// TIA Portal project "S71200OPCUA" (V16)

(* hardware
DEVICE "S7-1200 station_1"  S7-1200 Station
   slot 0: "Rack_0"  S7-1200 Rack  Rack  V1.0
   slot 1: "PLC_1"  CPU 1212C AC/DC/Rly  6ES7 212-1BE40-0XB0  V4.4
*)

// ===== PLC "PLC_1"  CPU 1212C AC/DC/Rly =====

VAR_GLOBAL   // PLC tag table "Default tag table"
   "Clock_Byte" AT %MB0 : Byte;
   "Clock_10Hz" AT %M0.0 : Bool;
   "Clock_5Hz" AT %M0.1 : Bool;
   "Clock_2.5Hz" AT %M0.2 : Bool;
   "Clock_2Hz" AT %M0.3 : Bool;
   "Clock_1.25Hz" AT %M0.4 : Bool;
   "Clock_1Hz" AT %M0.5 : Bool;
   "Clock_0.625Hz" AT %M0.6 : Bool;
   "Clock_0.5Hz" AT %M0.7 : Bool;
   "Disconnect" AT %M10.0 : Bool;
   "I_Sensor" AT %I10.0 : Bool;
   "Q_Speed" AT %QD100 : Real;
   "I_Boxdetected" AT %I10.1 : Bool;
   "I_PosX" AT %ID100 : Real;
   "I_PosY" AT %ID104 : Real;
   "I_PosZ" AT %ID108 : Real;
   "Q_PosX" AT %QD104 : Real;
   "Q_PosY" AT %QD108 : Real;
   "Q_PosZ" AT %QD112 : Real;
   "Q_Vacuum" AT %Q10.0 : Bool;
   "I_Flow" AT %ID112 : Real;
   "I_Level" AT %ID116 : Real;
   "Q_Filling" AT %QD116 : Real;
   "Q_Draining" AT %QD120 : Real;
   "I_Diffuse2m(1)" AT %I10.2 : Bool;
   "I_Diffuse2m(2)" AT %I10.3 : Bool;
   "Q_Conveyor2m(1)" AT %Q10.1 : Bool;
   "Q_Conveyor2m(2)" AT %Q10.2 : Bool;
END_VAR

DATA_BLOCK "OPC"   // DB1
{ S7_Optimized_Access := 'TRUE' }
VERSION : 0.1
   VAR
      Tank : Struct
         I_Level : Real;
         I_Flow : Real;
         Q_Filling : Real;
         Q_Draining : Real;
      END_STRUCT;
      Conveyor : Struct
         Q_Conveyor : Bool;
         "I_Sensor2m(1)" : Bool;
         "I_Sensor2m(2)" : Bool;
         "Q_Conveyor2m(1)" : Bool;
         "Q_Conveyor2m(2)" : Bool;
         I_Start : Bool;
         I_Stop : Bool;
         Q_Speed : Real;
         I_Sensor : Bool;
         Q_BoxCount : DInt;
         I_Reset : Bool;
         I_Maxlimit : Real := 6.0;
         I_Minlimit : Real := 2.0;
         I_Speed : Real := 1.0;
      END_STRUCT;
      "Pick and Place axis" : Struct
         I_Tolerance : Real := 0.02;
         IQ_Step : Int;
         I_Start : Bool;
         I_Init : Bool;
         I_XPos : Real;
         I_YPos : Real;
         I_ZPos : Real;
         I_BoxDetect : Bool;
         Q_XPos : Real;
         Q_YPos : Real;
         Q_ZPos : Real;
         Q_Vacuum : Bool;
         Q_Placed : Bool;
         Pos1 : Struct
            X : Real := 2.7;
            Y : Real := 3.9;
            Z : Real := 5.0;
         END_STRUCT;
         Pos2 : Struct
            X : Real := 6.6;
            Y : Real := 3.3;
            Z : Real := 4.2;
         END_STRUCT;
      END_STRUCT;
      Process : Struct
         I_Start : Bool;
         I_Stop : Bool;
         Process : Bool;
      END_STRUCT;
   END_VAR
BEGIN
END_DATA_BLOCK

// folder: 3Axis

DATA_BLOCK "Axis_DB"   // DB4
{ S7_Optimized_Access := 'TRUE' }
VERSION : 0.1
// stored: InstanceOfName Axis
"Axis"
BEGIN
END_DATA_BLOCK

// folder: Conveyor

DATA_BLOCK "IEC_Counter_0_DB"   // DB2
{ S7_Optimized_Access := 'TRUE' }
AUTHOR : Simatic
FAMILY : IEC
NAME : CNTR
VERSION : 1.0
// stored: InstanceOfName IEC_COUNTER
"IEC_COUNTER"
BEGIN
END_DATA_BLOCK

DATA_BLOCK "Conveyor_DB_1"   // DB5
{ S7_Optimized_Access := 'TRUE' }
VERSION : 0.1
// stored: InstanceOfName Conveyor
"Conveyor"
BEGIN
END_DATA_BLOCK

// folder: System blocks/Program resources

DATA_BLOCK "IEC_Timer_0_DB_1"   // DB3
{ S7_Optimized_Access := 'TRUE' }
AUTHOR : Simatic
FAMILY : IEC
NAME : IEC_TMR
VERSION : 1.0
// stored: InstanceOfName IEC_TIMER
"IEC_TIMER"
BEGIN
END_DATA_BLOCK

DATA_BLOCK "IEC_Timer_0_DB"   // DB6
{ S7_Optimized_Access := 'TRUE' }
AUTHOR : Simatic
FAMILY : IEC
NAME : IEC_TMR
VERSION : 1.0
// stored: InstanceOfName IEC_TIMER
"IEC_TIMER"
BEGIN
END_DATA_BLOCK

DATA_BLOCK "IEC_Timer_0_DB_2"   // DB7
{ S7_Optimized_Access := 'TRUE' }
AUTHOR : Simatic
FAMILY : IEC
NAME : IEC_TMR
VERSION : 1.0
// stored: InstanceOfName IEC_TIMER
"IEC_TIMER"
BEGIN
END_DATA_BLOCK

// folder: (top level)

ORGANIZATION_BLOCK "Main"   // OB1, FBD, ProgramCycle
TITLE = "Main Program Sweep (Cycle)"
{ S7_Optimized_Access := 'TRUE' }
VERSION : 0.1
   VAR_INPUT
      Initial_Call : Bool;   // Initial call of this OB
      Remanence : Bool;   // =True, if remanent data are available
   END_VAR
BEGIN

REGION Network 1: Process
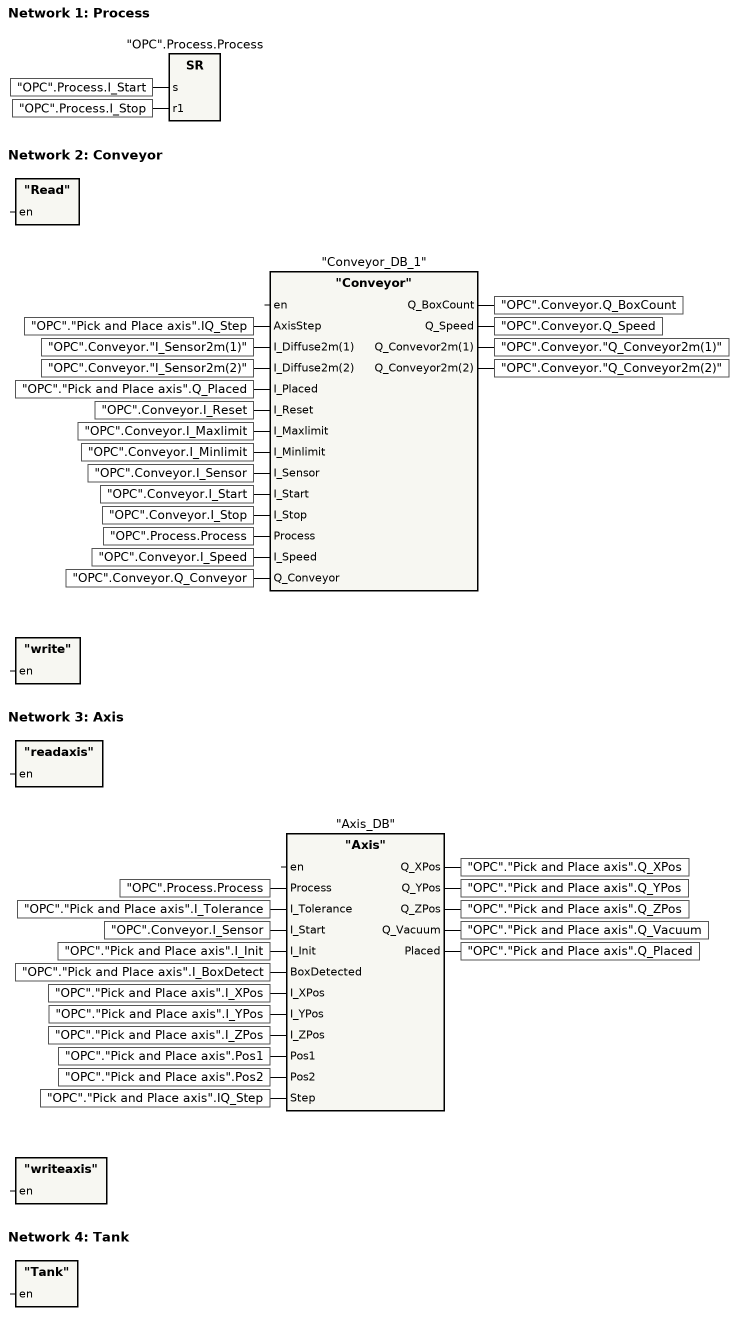
   IF "OPC".Process.I_Start THEN
       "OPC".Process.Process := TRUE;   // SR flip-flop
   END_IF;
   IF "OPC".Process.I_Stop THEN "OPC".Process.Process := FALSE; END_IF;
END_REGION

REGION Network 2: Conveyor
   "Read"();
   "Conveyor_DB_1"(AxisStep := "OPC"."Pick and Place axis".IQ_Step,   // "Conveyor"
                   "I_Diffuse2m(1)" := "OPC".Conveyor."I_Sensor2m(1)",
                   "I_Diffuse2m(2)" := "OPC".Conveyor."I_Sensor2m(2)",
                   I_Placed := "OPC"."Pick and Place axis".Q_Placed,
                   I_Reset := "OPC".Conveyor.I_Reset,
                   I_Maxlimit := "OPC".Conveyor.I_Maxlimit,
                   I_Minlimit := "OPC".Conveyor.I_Minlimit,
                   I_Sensor := "OPC".Conveyor.I_Sensor,
                   I_Start := "OPC".Conveyor.I_Start,
                   I_Stop := "OPC".Conveyor.I_Stop,
                   Process := "OPC".Process.Process,
                   I_Speed := "OPC".Conveyor.I_Speed,
                   Q_Conveyor := "OPC".Conveyor.Q_Conveyor,
                   Q_BoxCount => "OPC".Conveyor.Q_BoxCount,
                   Q_Speed => "OPC".Conveyor.Q_Speed,
                   "Q_Convevor2m(1)" => "OPC".Conveyor."Q_Conveyor2m(1)",
                   "Q_Conveyor2m(2)" => "OPC".Conveyor."Q_Conveyor2m(2)");
   "write"();
END_REGION

REGION Network 3: Axis
   "readaxis"();
   "Axis_DB"(Process := "OPC".Process.Process,   // "Axis"
             I_Tolerance := "OPC"."Pick and Place axis".I_Tolerance,
             I_Start := "OPC".Conveyor.I_Sensor,
             I_Init := "OPC"."Pick and Place axis".I_Init,
             BoxDetected := "OPC"."Pick and Place axis".I_BoxDetect,
             I_XPos := "OPC"."Pick and Place axis".I_XPos,
             I_YPos := "OPC"."Pick and Place axis".I_YPos,
             I_ZPos := "OPC"."Pick and Place axis".I_ZPos,
             Pos1 := "OPC"."Pick and Place axis".Pos1,
             Pos2 := "OPC"."Pick and Place axis".Pos2,
             "Step" := "OPC"."Pick and Place axis".IQ_Step,
             Q_XPos => "OPC"."Pick and Place axis".Q_XPos,
             Q_YPos => "OPC"."Pick and Place axis".Q_YPos,
             Q_ZPos => "OPC"."Pick and Place axis".Q_ZPos,
             Q_Vacuum => "OPC"."Pick and Place axis".Q_Vacuum,
             Placed => "OPC"."Pick and Place axis".Q_Placed);
   "writeaxis"();
END_REGION

REGION Network 4: Tank
   "Tank"();
END_REGION
END_ORGANIZATION_BLOCK

// folder: 3Axis

FUNCTION_BLOCK "Axis"   // FB3, FBD
{ S7_Optimized_Access := 'TRUE' }
VERSION : 0.1
   VAR_INPUT
      Process : Bool;
      I_Tolerance : Real;
      I_Start : Bool;
      I_Init : Bool;
      BoxDetected : Bool;
      I_XPos : Real;
      I_YPos : Real;
      I_ZPos : Real;
      Pos1 : Struct
         X : Real;
         Y : Real;
         Z : Real;
      END_STRUCT;
      Pos2 : Struct
         X : Real;
         Y : Real;
         Z : Real;
      END_STRUCT;
   END_VAR
   VAR_OUTPUT
      Q_XPos : Real;
      Q_YPos : Real;
      Q_ZPos : Real;
      Q_Vacuum : Bool;
      Placed : Bool;
   END_VAR
   VAR_IN_OUT
      "Step" : Int;
   END_VAR
   VAR
      PosX1Min : Real;
      PosX1Max : Real;
      PosY1Min : Real;
      PosY1Max : Real;
      PosZ1Min : Real;
      PosZ1Max : Real;
      PosX2Min : Real;
      PosX2Max : Real;
      PosY2Min : Real;
      PosY2Max : Real;
      PosZ2Min : Real;
      PosZ2Max : Real;
   END_VAR
   VAR_TEMP   // added for the SCL form of the ladder/FBD networks
      _w1 : Bool;
   END_VAR
BEGIN

REGION Network 1: Position Tolerance P1
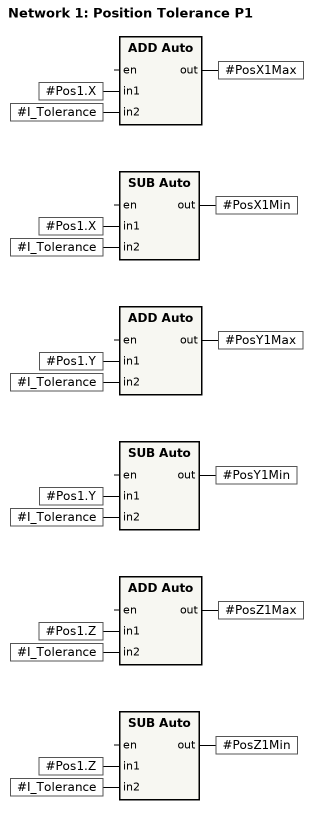
   #PosX1Max := #Pos1.X + #I_Tolerance;
   #PosX1Min := #Pos1.X - #I_Tolerance;
   #PosY1Max := #Pos1.Y + #I_Tolerance;
   #PosY1Min := #Pos1.Y - #I_Tolerance;
   #PosZ1Max := #Pos1.Z + #I_Tolerance;
   #PosZ1Min := #Pos1.Z - #I_Tolerance;
END_REGION

REGION Network 2: Position Tolerance P2
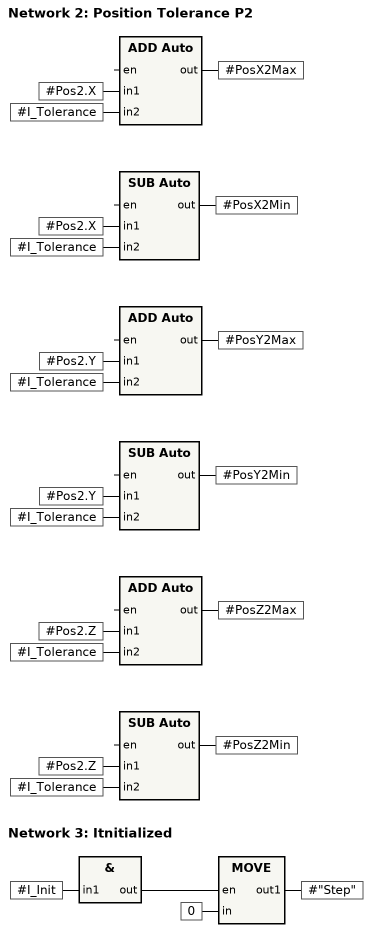
   #PosX2Max := #Pos2.X + #I_Tolerance;
   #PosX2Min := #Pos2.X - #I_Tolerance;
   #PosY2Max := #Pos2.Y + #I_Tolerance;
   #PosY2Min := #Pos2.Y - #I_Tolerance;
   #PosZ2Max := #Pos2.Z + #I_Tolerance;
   #PosZ2Min := #Pos2.Z - #I_Tolerance;
END_REGION

REGION Network 3: Itnitialized
   IF #I_Init THEN #"Step" := 0; END_IF;
END_REGION

REGION Network 4: Cycle
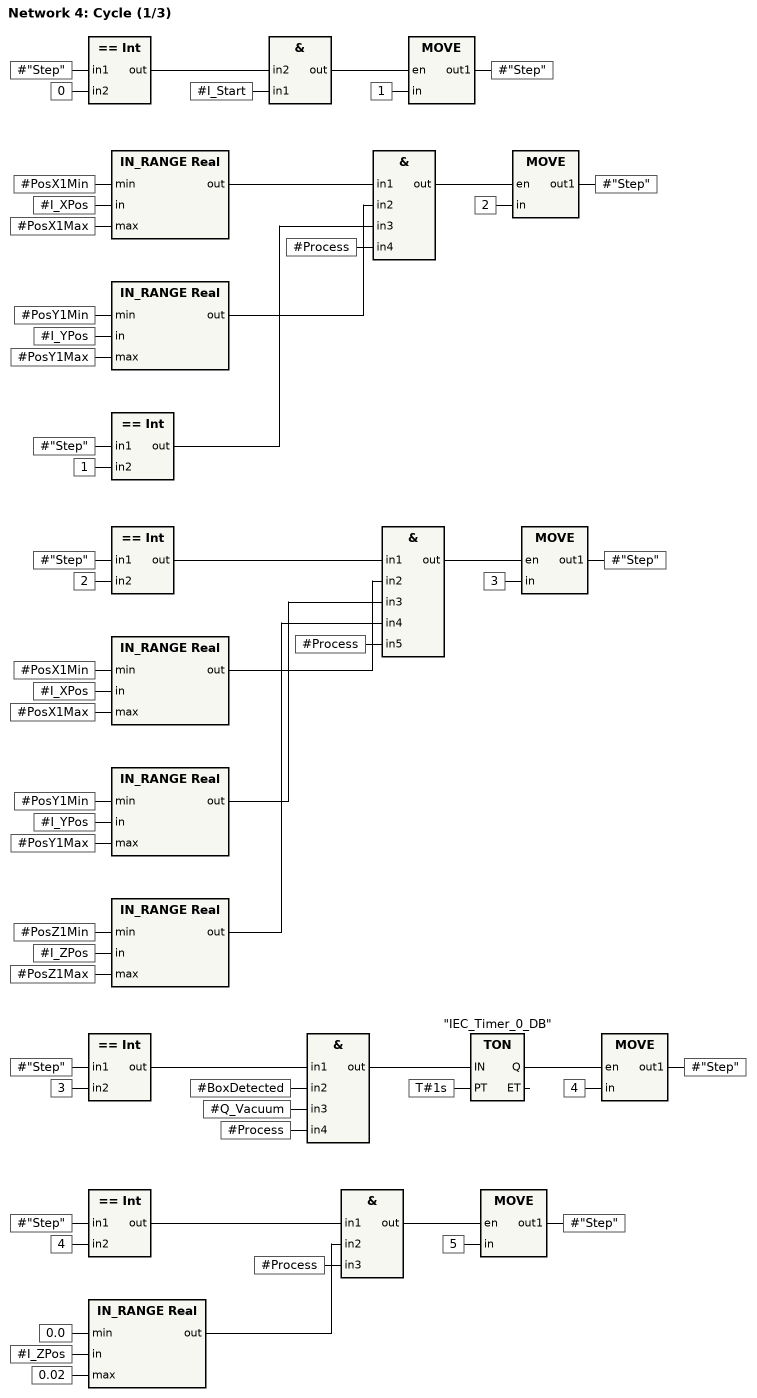
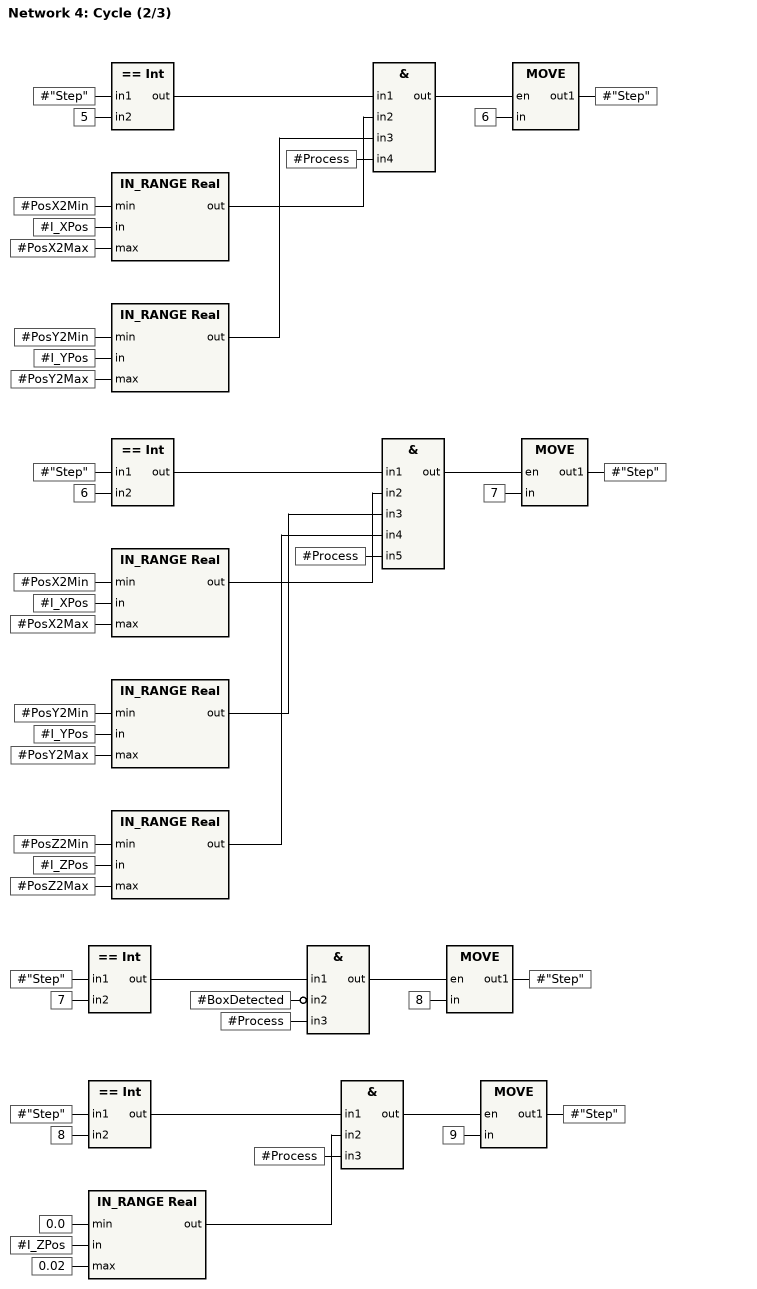
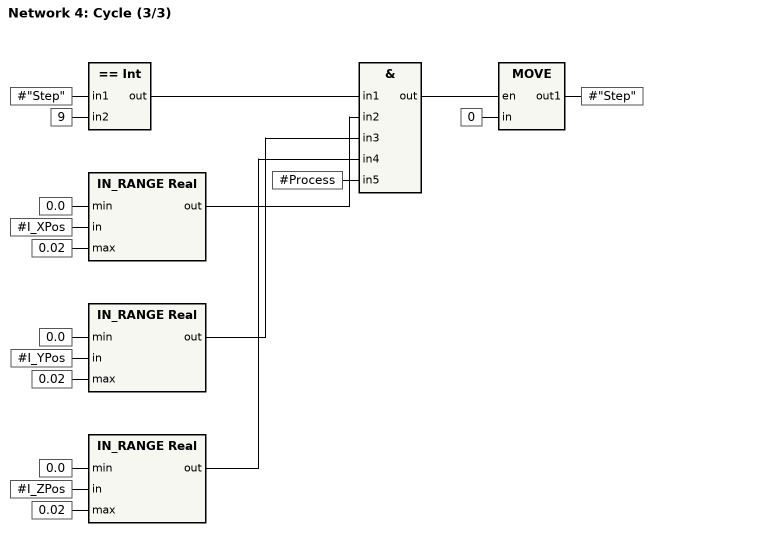
   IF (#"Step" = 0) AND #I_Start THEN #"Step" := 1; END_IF;
   IF (#PosX1Min <= #I_XPos) AND (#I_XPos <= #PosX1Max) AND (#PosY1Min <= #I_YPos) AND (#I_YPos <= #PosY1Max) AND (#"Step" = 1) AND #Process THEN
       #"Step" := 2;
   END_IF;
   IF (#"Step" = 2) AND (#PosX1Min <= #I_XPos) AND (#I_XPos <= #PosX1Max) AND (#PosY1Min <= #I_YPos) AND (#I_YPos <= #PosY1Max) AND (#PosZ1Min <= #I_ZPos) AND (#I_ZPos <= #PosZ1Max) AND #Process THEN
       #"Step" := 3;
   END_IF;
   "IEC_Timer_0_DB".TON(IN := (#"Step" = 3) AND #BoxDetected AND #Q_Vacuum AND #Process, PT := T#1s);
   IF "IEC_Timer_0_DB".Q THEN #"Step" := 4; END_IF;
   IF (#"Step" = 4) AND (0.0 <= #I_ZPos) AND (#I_ZPos <= 0.02) AND #Process THEN #"Step" := 5; END_IF;
   IF (#"Step" = 5) AND (#PosX2Min <= #I_XPos) AND (#I_XPos <= #PosX2Max) AND (#PosY2Min <= #I_YPos) AND (#I_YPos <= #PosY2Max) AND #Process THEN
       #"Step" := 6;
   END_IF;
   IF (#"Step" = 6) AND (#PosX2Min <= #I_XPos) AND (#I_XPos <= #PosX2Max) AND (#PosY2Min <= #I_YPos) AND (#I_YPos <= #PosY2Max) AND (#PosZ2Min <= #I_ZPos) AND (#I_ZPos <= #PosZ2Max) AND #Process THEN
       #"Step" := 7;
   END_IF;
   IF (#"Step" = 7) AND NOT #BoxDetected AND #Process THEN #"Step" := 8; END_IF;
   IF (#"Step" = 8) AND (0.0 <= #I_ZPos) AND (#I_ZPos <= 0.02) AND #Process THEN #"Step" := 9; END_IF;
   IF (#"Step" = 9) AND (0.0 <= #I_XPos) AND (#I_XPos <= 0.02) AND (0.0 <= #I_YPos) AND (#I_YPos <= 0.02) AND (0.0 <= #I_ZPos) AND (#I_ZPos <= 0.02) AND #Process THEN
       #"Step" := 0;
   END_IF;
END_REGION

REGION Network 5: Execution
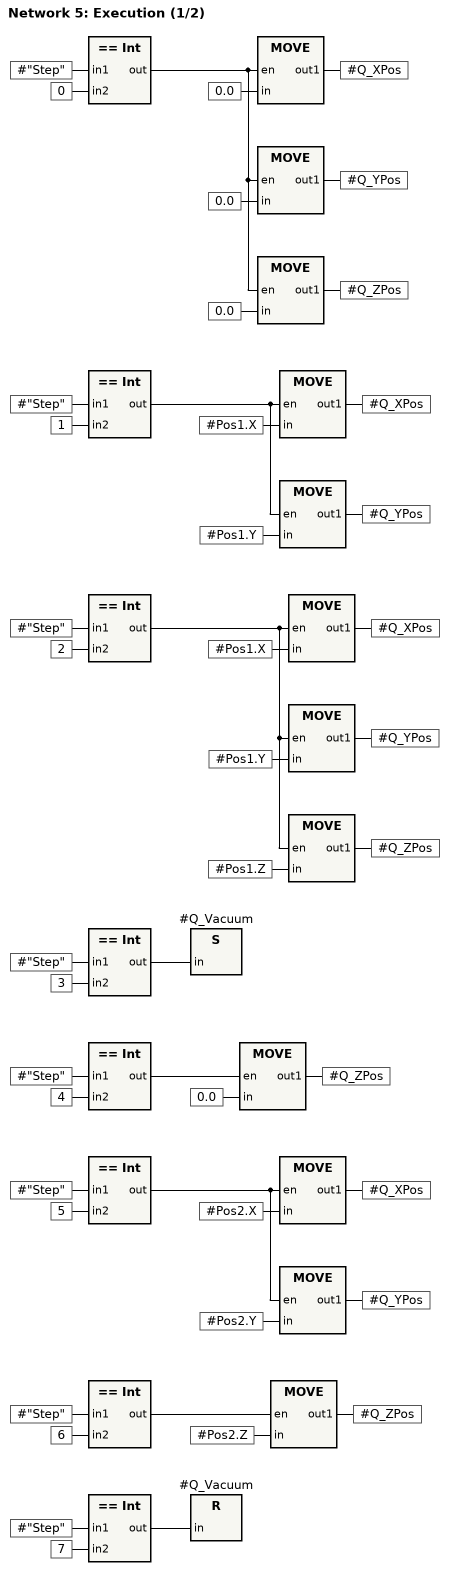
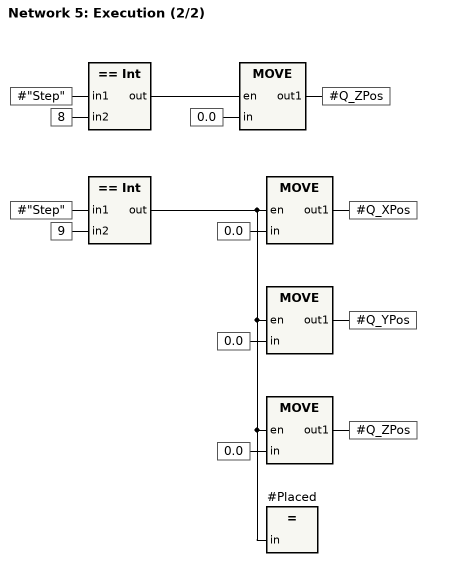
   IF #"Step" = 0 THEN
       #Q_XPos := 0.0;
       #Q_YPos := 0.0;
       #Q_ZPos := 0.0;
   END_IF;
   IF #"Step" = 1 THEN
       #Q_XPos := #Pos1.X;
       #Q_YPos := #Pos1.Y;
   END_IF;
   IF #"Step" = 2 THEN
       #Q_XPos := #Pos1.X;
       #Q_YPos := #Pos1.Y;
       #Q_ZPos := #Pos1.Z;
   END_IF;
   IF #"Step" = 3 THEN #Q_Vacuum := TRUE; END_IF;
   IF #"Step" = 4 THEN #Q_ZPos := 0.0; END_IF;
   IF #"Step" = 5 THEN
       #Q_XPos := #Pos2.X;
       #Q_YPos := #Pos2.Y;
   END_IF;
   IF #"Step" = 6 THEN #Q_ZPos := #Pos2.Z; END_IF;
   IF #"Step" = 7 THEN #Q_Vacuum := FALSE; END_IF;
   IF #"Step" = 8 THEN #Q_ZPos := 0.0; END_IF;
   #_w1 := #"Step" = 9;
   IF #_w1 THEN
       #Q_XPos := 0.0;
       #Q_YPos := 0.0;
       #Q_ZPos := 0.0;
   END_IF;
   #Placed := #_w1;
END_REGION
END_FUNCTION_BLOCK

FUNCTION "readaxis" : Void   // FC3, SCL
{ S7_Optimized_Access := 'TRUE' }
VERSION : 0.1
BEGIN
   "OPC"."Pick and Place axis".I_XPos := "I_PosX";
   "OPC"."Pick and Place axis".I_YPos  := "I_PosY";
   "OPC"."Pick and Place axis".I_ZPos := "I_PosZ";
   "OPC"."Pick and Place axis".I_BoxDetect := "I_Boxdetected";
END_FUNCTION

FUNCTION "writeaxis" : Void   // FC4, SCL
{ S7_Optimized_Access := 'TRUE' }
VERSION : 0.1
BEGIN
   "Q_PosX":=  "OPC"."Pick and Place axis".Q_XPos;
   "Q_PosY" :=  "OPC"."Pick and Place axis".Q_YPos ;
   "Q_PosZ" := "OPC"."Pick and Place axis".Q_ZPos ;
   "Q_Vacuum" :=  "OPC"."Pick and Place axis".Q_Vacuum ;
END_FUNCTION

// folder: Conveyor

FUNCTION_BLOCK "Conveyor"   // FB2, FBD
{ S7_Optimized_Access := 'TRUE' }
VERSION : 0.1
   VAR_INPUT
      AxisStep : Int;
      "I_Diffuse2m(1)" : Bool;
      "I_Diffuse2m(2)" : Bool;
      I_Placed : Bool;
      I_Reset : Bool;
      I_Maxlimit : Real;
      I_Minlimit : Real;
      I_Sensor : Bool;
      I_Start : Bool;
      I_Stop : Bool;
      Process : Bool;
   END_VAR
   VAR_OUTPUT
      Q_BoxCount : DInt;
      Q_Speed : Real;
      "Q_Convevor2m(1)" : Bool;
      "Q_Conveyor2m(2)" : Bool;
   END_VAR
   VAR_IN_OUT
      I_Speed : Real;
      Q_Conveyor : Bool;
   END_VAR
   VAR
      PulseR : Bool;
      PulseN : Bool;
   END_VAR
   VAR_TEMP   // added for the SCL form of the ladder/FBD networks
      _w1 : Bool;
      _w2 : Bool;
   END_VAR
BEGIN

REGION Network 1: Convevor Start-Stop
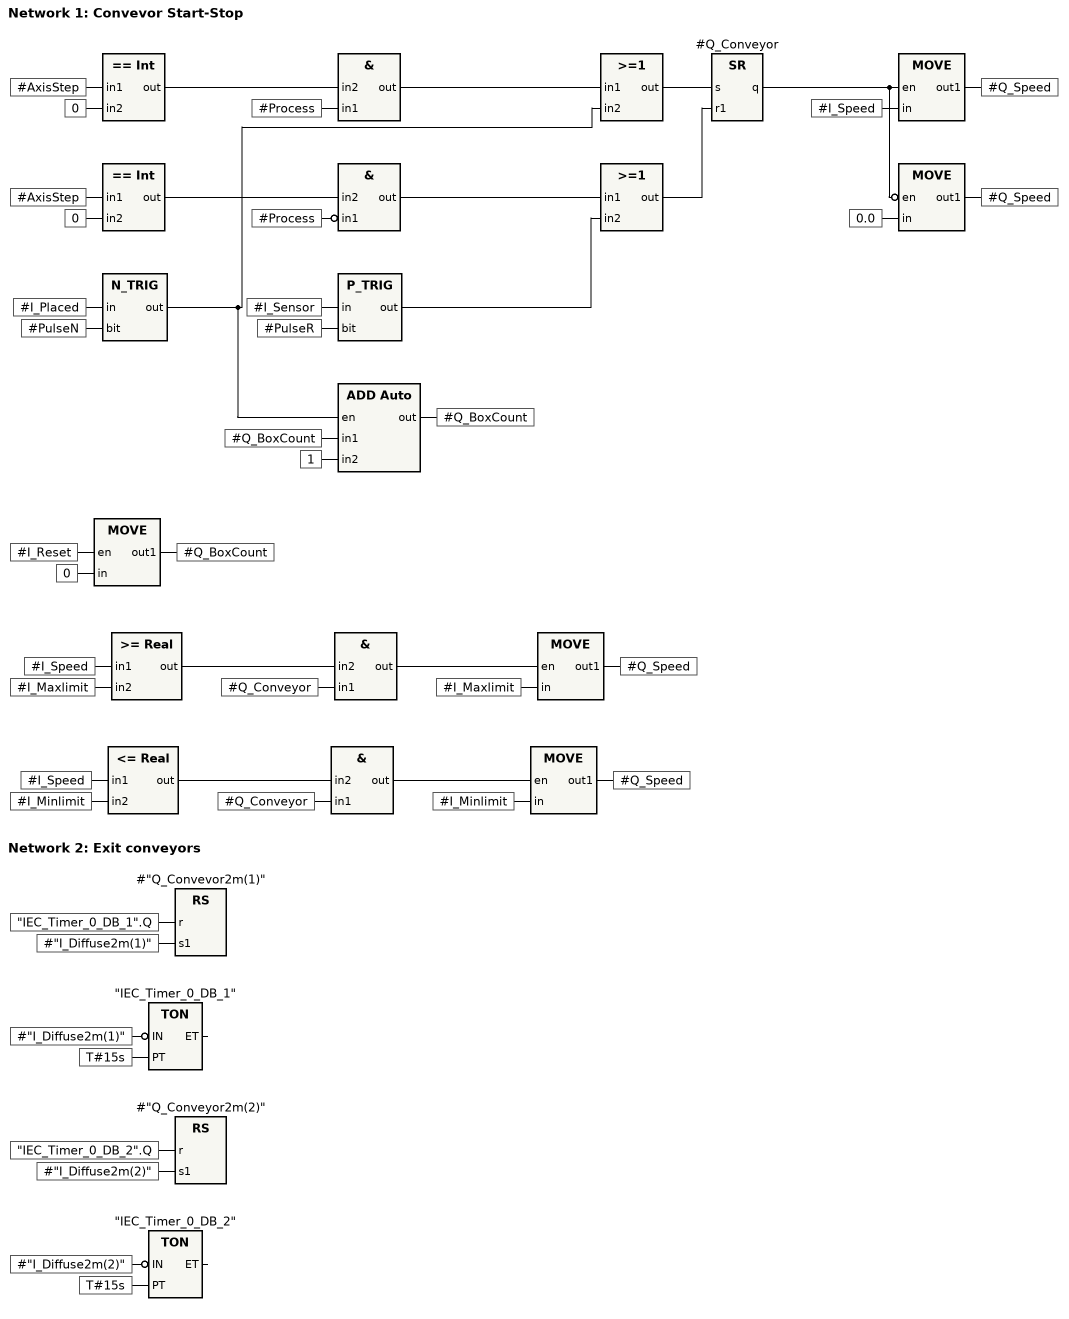
   #_w1 := NOT #I_Placed AND #PulseN;   // falling edge
   #PulseN := #I_Placed;
   #_w2 := #I_Sensor AND NOT #PulseR;   // rising edge
   #PulseR := #I_Sensor;
   IF ((#AxisStep = 0) AND #Process) OR #_w1 THEN
       #Q_Conveyor := TRUE;   // SR flip-flop
   END_IF;
   IF ((#AxisStep = 0) AND NOT #Process) OR #_w2 THEN #Q_Conveyor := FALSE; END_IF;
   IF #Q_Conveyor THEN #Q_Speed := #I_Speed; END_IF;
   IF NOT #Q_Conveyor THEN #Q_Speed := 0.0; END_IF;
   IF #_w1 THEN #Q_BoxCount := #Q_BoxCount + 1; END_IF;
   IF #I_Reset THEN #Q_BoxCount := 0; END_IF;
   IF (#I_Speed >= #I_Maxlimit) AND #Q_Conveyor THEN #Q_Speed := #I_Maxlimit; END_IF;
   IF (#I_Speed <= #I_Minlimit) AND #Q_Conveyor THEN #Q_Speed := #I_Minlimit; END_IF;
END_REGION

REGION Network 2: Exit conveyors
   IF "IEC_Timer_0_DB_1".Q THEN
       #"Q_Convevor2m(1)" := FALSE;   // RS flip-flop
   END_IF;
   IF #"I_Diffuse2m(1)" THEN #"Q_Convevor2m(1)" := TRUE; END_IF;
   "IEC_Timer_0_DB_1".TON(IN := NOT #"I_Diffuse2m(1)", PT := T#15s);
   IF "IEC_Timer_0_DB_2".Q THEN
       #"Q_Conveyor2m(2)" := FALSE;   // RS flip-flop
   END_IF;
   IF #"I_Diffuse2m(2)" THEN #"Q_Conveyor2m(2)" := TRUE; END_IF;
   "IEC_Timer_0_DB_2".TON(IN := NOT #"I_Diffuse2m(2)", PT := T#15s);
END_REGION
END_FUNCTION_BLOCK

FUNCTION "Read" : Void   // FC1, SCL
{ S7_Optimized_Access := 'TRUE' }
VERSION : 0.1
BEGIN
   "OPC".Conveyor.I_Sensor := "I_Sensor";
   "OPC".Conveyor."I_Sensor2m(1)" := "I_Diffuse2m(1)";
   "OPC".Conveyor."I_Sensor2m(2)" := "I_Diffuse2m(2)";
END_FUNCTION

FUNCTION "write" : Void   // FC2, SCL
{ S7_Optimized_Access := 'TRUE' }
VERSION : 0.1
BEGIN
   "Q_Speed" := "OPC".Conveyor.Q_Speed;
   "Q_Conveyor2m(1)" := "OPC".Conveyor."Q_Conveyor2m(1)";
   "Q_Conveyor2m(2)" := "OPC".Conveyor."Q_Conveyor2m(2)";
END_FUNCTION

// folder: Tank

FUNCTION "Tank" : Void   // FC5, SCL
{ S7_Optimized_Access := 'TRUE' }
VERSION : 0.1
BEGIN
   "Q_Filling" := "OPC".Tank.Q_Filling;
   "Q_Draining" := "OPC".Tank.Q_Draining;

   "OPC".Tank.I_Level:= "I_Level";
   "OPC".Tank.I_Flow :="I_Flow" ;
END_FUNCTION